PROGRAM GL3_Accumulation
VAR
	
	RUN_FWD_TO_GL4_BIT : BOOL; // GL4 EMPTY SO SEND PART FROM GL3 TO GL4
	RUN_FWD_TO_EXIT_BIT : BOOL; // RUN GL3 FWD TO EXIT SENSOR
	GL4_ENTRY_FTRIG:  F_TRIG;
	
END_VAR
VAR // added by the converter: edge detectors and wires of the graphical bodies
    _w1 : BOOL;
END_VAR

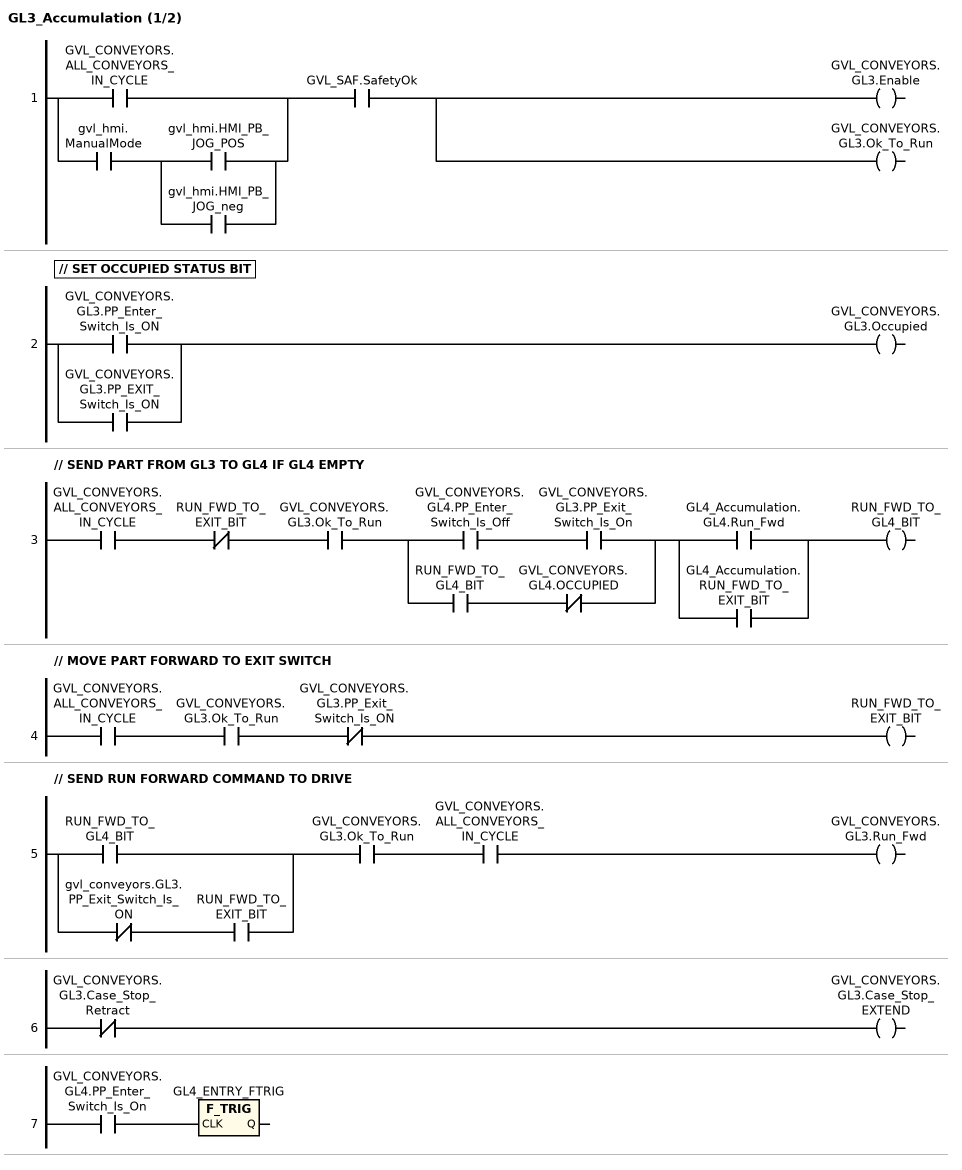
// NETWORK 1
_w1 := (GVL_CONVEYORS.ALL_CONVEYORS_IN_CYCLE OR gvl_hmi.ManualMode AND (gvl_hmi.HMI_PB_JOG_POS OR gvl_hmi.HMI_PB_JOG_neg)) AND GVL_SAF.SafetyOk;
GVL_CONVEYORS.GL3.Enable := _w1;
GVL_CONVEYORS.GL3.Ok_To_Run := _w1;

// NETWORK 2
// label: // SET OCCUPIED STATUS BIT
GVL_CONVEYORS.GL3.Occupied := GVL_CONVEYORS.GL3.PP_Enter_Switch_Is_ON OR GVL_CONVEYORS.GL3.PP_EXIT_Switch_Is_ON;

// NETWORK 3: // SEND PART FROM GL3 TO GL4 IF GL4 EMPTY
RUN_FWD_TO_GL4_BIT := GVL_CONVEYORS.ALL_CONVEYORS_IN_CYCLE AND NOT RUN_FWD_TO_EXIT_BIT AND GVL_CONVEYORS.GL3.Ok_To_Run AND (GVL_CONVEYORS.GL4.PP_Enter_Switch_Is_Off AND GVL_CONVEYORS.GL3.PP_Exit_Switch_Is_On OR RUN_FWD_TO_GL4_BIT AND NOT GVL_CONVEYORS.GL4.OCCUPIED) AND (GL4_Accumulation.GL4.Run_Fwd OR GL4_Accumulation.RUN_FWD_TO_EXIT_BIT);

// NETWORK 4: // MOVE PART FORWARD TO EXIT SWITCH
RUN_FWD_TO_EXIT_BIT := GVL_CONVEYORS.ALL_CONVEYORS_IN_CYCLE AND GVL_CONVEYORS.GL3.Ok_To_Run AND NOT GVL_CONVEYORS.GL3.PP_Exit_Switch_Is_ON;

// NETWORK 5: // SEND RUN FORWARD COMMAND TO DRIVE
GVL_CONVEYORS.GL3.Run_Fwd := (RUN_FWD_TO_GL4_BIT OR NOT gvl_conveyors.GL3.PP_Exit_Switch_Is_ON AND RUN_FWD_TO_EXIT_BIT) AND GVL_CONVEYORS.GL3.Ok_To_Run AND GVL_CONVEYORS.ALL_CONVEYORS_IN_CYCLE;

// NETWORK 6
GVL_CONVEYORS.GL3.Case_Stop_EXTEND := NOT GVL_CONVEYORS.GL3.Case_Stop_Retract;

// NETWORK 7
GL4_ENTRY_FTRIG(CLK := GVL_CONVEYORS.GL4.PP_Enter_Switch_Is_On); // F_TRIG

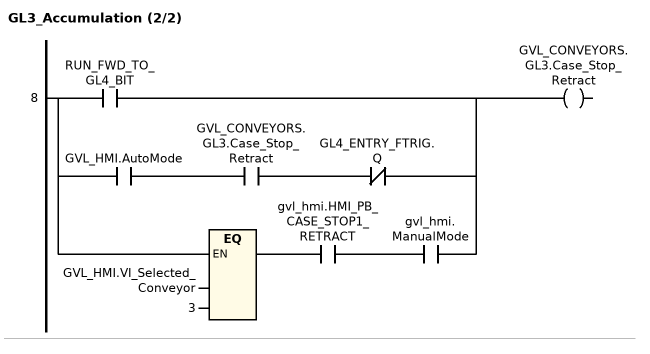
// NETWORK 8
GVL_CONVEYORS.GL3.Case_Stop_Retract := RUN_FWD_TO_GL4_BIT OR GVL_HMI.AutoMode AND GVL_CONVEYORS.GL3.Case_Stop_Retract AND NOT GL4_ENTRY_FTRIG.Q OR GVL_HMI.VI_Selected_Conveyor = 3 AND gvl_hmi.HMI_PB_CASE_STOP1_RETRACT AND gvl_hmi.ManualMode;

END_PROGRAM

(* stored: Version 1.1.0.1, ProductVersion 3.1.4024.12
   POU GL3_Accumulation: Id {67906925-41d1-4f67-82c4-0ccfa49f7750}, SpecialFunc None *)
